// Mitsubishi GX Works2 project: 电动机正反转   PLC: FX1S

PROGRAM MAIN
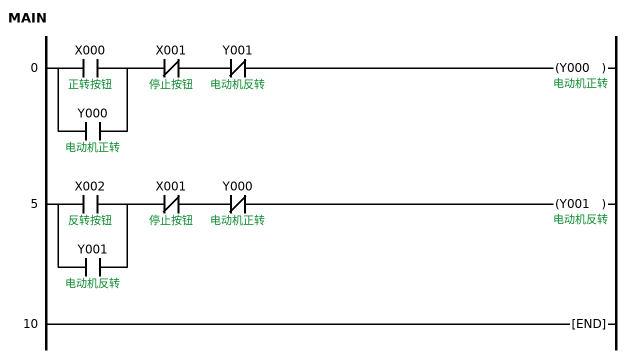
0     LD      X000  ; 正转按钮
      OR      Y000  ; 电动机正转
      ANI     X001  ; 停止按钮
      ANI     Y001  ; 电动机反转
      OUT     Y000  ; 电动机正转
5     LD      X002  ; 反转按钮
      OR      Y001  ; 电动机反转
      ANI     X001  ; 停止按钮
      ANI     Y000  ; 电动机正转
      OUT     Y001  ; 电动机反转
10    END
END_PROGRAM
